{attribute 'GeneratedUsingTerminal: AT2050-0500-0022'}
{attribute addProperty BoxType "AT2050-0500-0022"}
{attribute addProperty Id "A_0091_AT2020_5250_0017_AT2020_5250AT2020_33A3DF1B80"}
{attribute addProperty CRC "1127996926"}
{attribute addProperty Size "80"}
TYPE A_0053_AT2050_0500_0022_433BDDFE EXTENDS AT2050_A7FEA1CF :
STRUCT
	{attribute addProperty Name "A_0091_AT2020_5250_0017_AT2020_5250"}
	{attribute addProperty PreviousPort "A_0053(AT2050-0500-0022) : B"}
	A_0091_AT2020_5250_0017_AT2020_5250 : AT2020_33A3DF1B;
END_STRUCT
END_TYPE

(* stored: Version 1.2.0.0, ProductVersion 3.1.4024.9
   DUT A_0053_AT2050_0500_0022_433BDDFE: Id {91b0921e-ae6d-46e8-9449-bfb9870f98b6} *)
